// CRC-32/ISO-HDLC over the record except its final CRC field (F_Crc32).
FUNCTION F_TcWindowsClockCrc : DWORD
VAR_INPUT
    Sample : ST_TcWindowsClockSampleV1;
END_VAR

F_TcWindowsClockCrc := F_Crc32(pData := ADR(Sample),
    Size := SIZEOF(Sample) - SIZEOF(Sample.Crc));

END_FUNCTION

(* stored: Version 1.1.0.1, ProductVersion 3.1.4024.12
   POU F_TcWindowsClockCrc: Id {7b4f1648-51cc-4f31-8ec7-202761708e8c}, SpecialFunc None *)
